(* Logix 5000 project; controller testing vendor 1 type 14 code 151 rev 32.11; software revision 32.00 *)

TASK MainTask (continuous, watchdog 500 ms) : MainProgram

MODULES
   Local : vendor 1 type 14 code 151 (Compact 0, rev 32.11)
      Analog_IO : Embedded (Compact 2, rev 1.1, Output RPI 80 ms)
      Counters : Embedded (Compact 3, rev 1.1, Output RPI 20 ms)
      Discrete_IO : Embedded (Compact 1, rev 3.1, Output RPI 20 ms)
END_MODULES

TYPE test :
STRUCT
   value1 : DINT;
   value2 : STRING;
   value3 : INT;
   value4 : BOOL;
   value5 : DINT[5];
END_STRUCT
END_TYPE

VAR_GLOBAL   (* controller tags *)
   string1 : STRING := 'testing1';
   string2 : STRING := 'testing2';
   string3 : STRING := 'testing3';
   string4 : STRING := 'testing4';
   string5 : STRING := 'testing5';
   string6 : STRING := 'testing6';
   string_array : STRING[5] := ([0] := 'testing2', [1] := 'testing3', [2] := 'testing4', [3] := 'testing5', [4] := 'testing6');
   stringread : STRING := 'testing1';
   test_array : DINT[5] := ([0] := 345, [1] := 5665, [2] := 341, [3] := 113121, [4] := 121314);
   udt_Item : test := (value1 := 367, value2 := 'testing2', value3 := 1200, value4 := 1, value5[0] := 6333, value5[1] := 923);
END_VAR

PROGRAM MainProgram   (* main routine MainRoutine *)
VAR
   Send_data : BOOL := 1;
END_VAR

ROUTINE MainRoutine   (* ladder *)
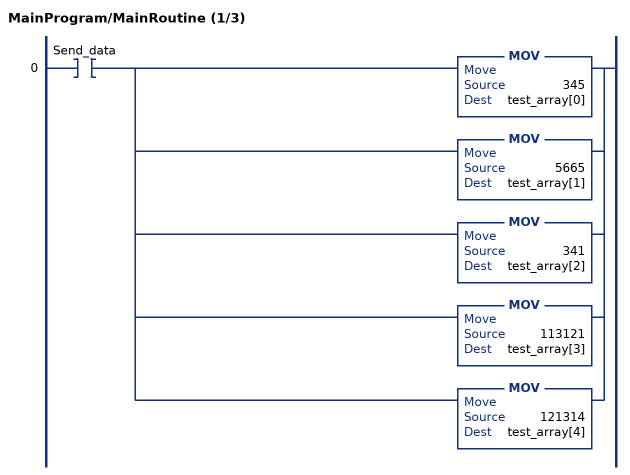
   0: XIC(Send_data)[MOV(345,test_array[0]) ,MOV(5665,test_array[1]) ,MOV(341,test_array[2]) ,MOV(113121,test_array[3]) ,MOV(121314,test_array[4]) ];
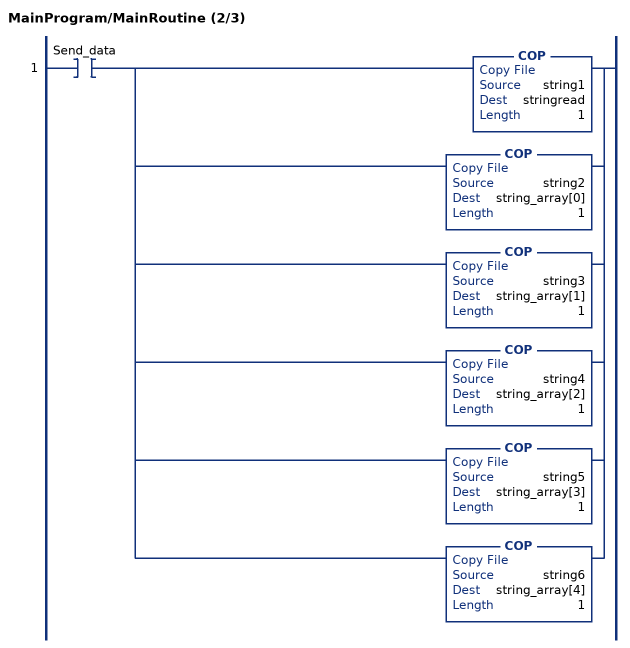
   1: XIC(Send_data)[COP(string1,stringread,1) ,COP(string2,string_array[0],1) ,COP(string3,string_array[1],1) ,COP(string4,string_array[2],1) ,COP(string5,string_array[3],1) ,COP(string6,string_array[4],1) ];
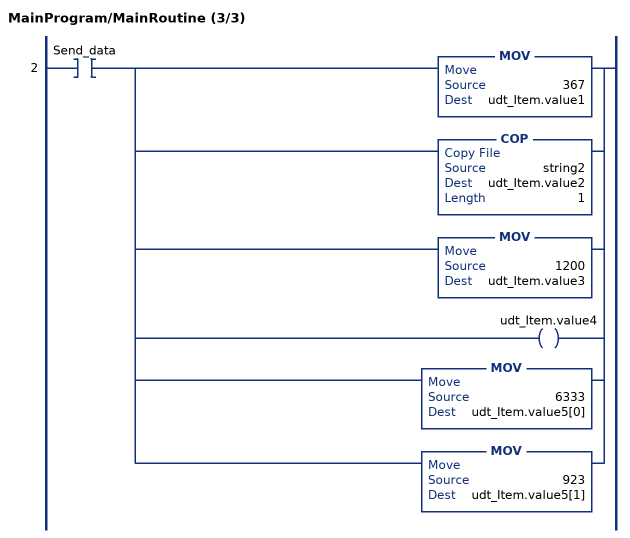
   2: XIC(Send_data)[MOV(367,udt_Item.value1) ,COP(string2,udt_Item.value2,1) ,MOV(1200,udt_Item.value3) ,OTE(udt_Item.value4) ,MOV(6333,udt_Item.value5[0]) ,MOV(923,udt_Item.value5[1]) ];
END_ROUTINE
END_PROGRAM
